// Mitsubishi GX Works2 project: 250627_단일공정순차제어(1)   PLC: Q02U

PROGRAM MAIN
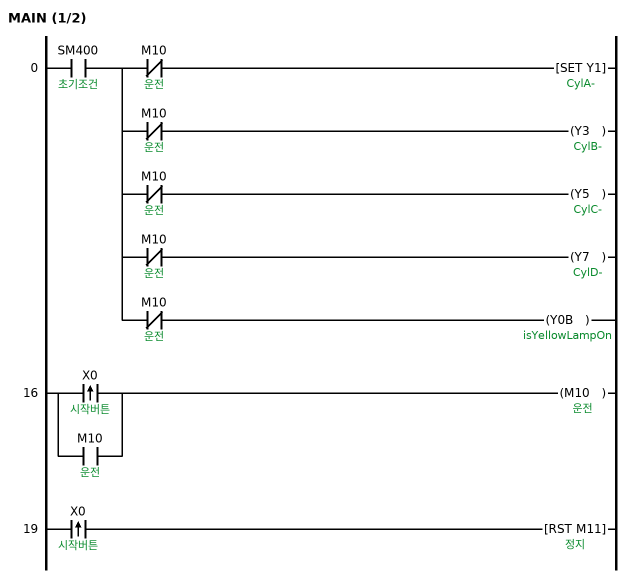
0     LD      SM400  ; 초기조건
      MPS
      ANI     M10  ; 운전
      SET     Y1  ; CylA-
      MRD
      ANI     M10  ; 운전
      OUT     Y3  ; CylB-
      MRD
      ANI     M10  ; 운전
      OUT     Y5  ; CylC-
      MRD
      ANI     M10  ; 운전
      OUT     Y7  ; CylD-
      MPP
      ANI     M10  ; 운전
      OUT     Y0B  ; isYellowLampOn
16    LDP     X0  ; 시작버튼
      OR      M10  ; 운전
      OUT     M10  ; 운전
19    LDP     X0  ; 시작버튼
      RST     M11  ; 정지
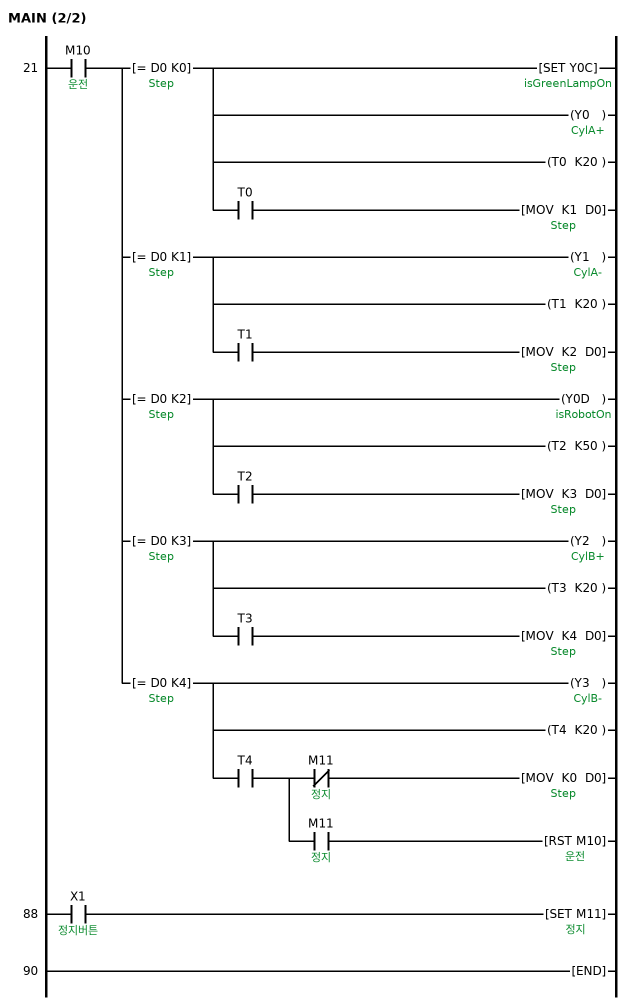
21    LD      M10  ; 운전
      MPS
      AND=    D0 K0  ; Step
      SET     Y0C  ; isGreenLampOn
      OUT     Y0  ; CylA+
      OUT     T0 K20
      AND     T0
      MOV     K1 D0
      MRD
      AND=    D0 K1  ; Step
      OUT     Y1  ; CylA-
      OUT     T1 K20
      AND     T1
      MOV     K2 D0
      MRD
      AND=    D0 K2  ; Step
      OUT     Y0D  ; isRobotOn
      OUT     T2 K50
      AND     T2
      MOV     K3 D0
      MRD
      AND=    D0 K3  ; Step
      OUT     Y2  ; CylB+
      OUT     T3 K20
      AND     T3
      MOV     K4 D0
      MPP
      AND=    D0 K4  ; Step
      OUT     Y3  ; CylB-
      OUT     T4 K20
      AND     T4
      MPS
      ANI     M11  ; 정지
      MOV     K0 D0
      MPP
      AND     M11  ; 정지
      RST     M10  ; 운전
88    LD      X1  ; 정지버튼
      SET     M11  ; 정지
90    END
END_PROGRAM

// device comments not shown above
X2  ; 긴급정지버튼
X19  ; 근접센서ON
X1A  ; 금속센서ON
Y4  ; CylC+
Y6  ; CylD+
Y8  ; isCW
Y9  ; isCCW
Y0A  ; isRedLampOn
